FUNCTION_BLOCK RepeatUnwrap IMPLEMENTS I_Unwrapper
VAR
	_x : UDINT;
	_y : UDINT;
END_VAR

METHOD Sample : BOOL
VAR_INPUT
	ImageWidth	: UDINT;
	ImageHeight	: UDINT;
	XOffset	: UDINT;
	YOffset	: UDINT;
END_VAR
_x	   := XOffset MOD (ImageWidth - 1);
_y	   := YOffset MOD (ImageHeight - 1);
Sample := TRUE;
END_METHOD

PROPERTY X : UDINT
GET
X := _x;
END_GET
END_PROPERTY

PROPERTY Y : UDINT
GET
Y := _y;
END_GET
END_PROPERTY

END_FUNCTION_BLOCK

(* stored: Version 1.1.0.1
   POU RepeatUnwrap: Id {fb22b2a3-89ed-4a06-98bf-5e65d51c49b6}, SpecialFunc None
   Method Sample: Id {ef543699-0062-41b2-961b-3cabad4dc6af}
   Property X: Id {3676239a-6f2b-42b2-9bff-c6e6ed30f39d}
   Get Get: Id {059c159d-bb18-439c-96e6-db3717d50c4c}
   Property Y: Id {3ff09c71-7c34-4d58-98f6-ae8c10a59a7e}
   Get Get: Id {e4b0ccd4-360e-48a6-a3c7-a51302a61789} *)
